REGION Network 51: Step[650] : Transfer PP Left Clamp Open
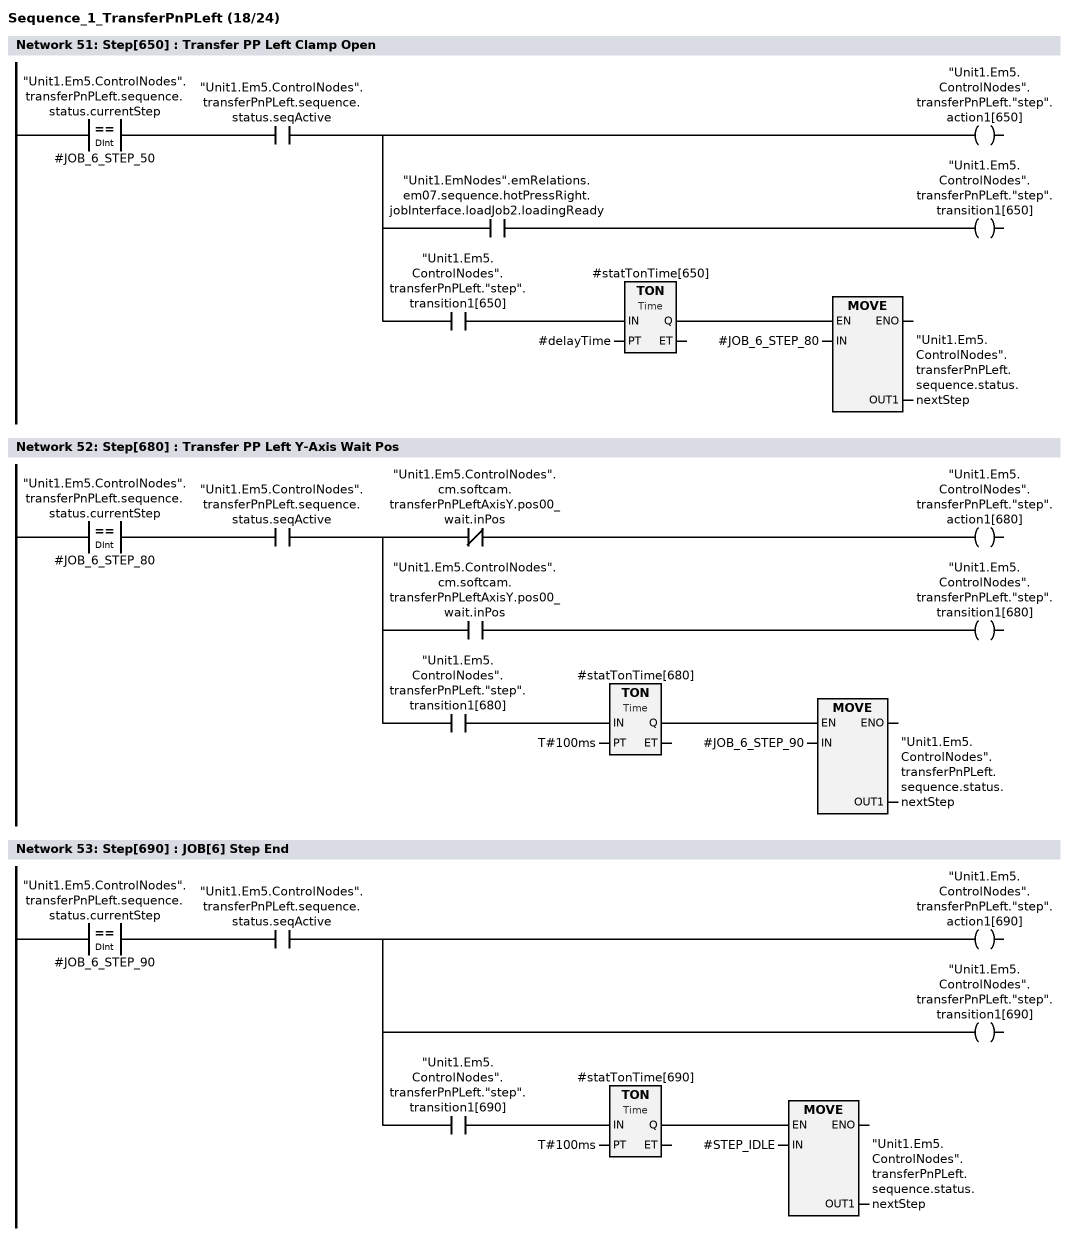
   RUNG wire#powerrail
      { S7_Templates := "SrcType := DInt" } EQ_Contact(in1 := "Unit1.Em5.ControlNodes".transferPnPLeft.sequence.status.currentStep, in2 := #JOB_6_STEP_50)
      Contact( "Unit1.Em5.ControlNodes".transferPnPLeft.sequence.status.seqActive )
      wire#w1
      Coil( "Unit1.Em5.ControlNodes".transferPnPLeft."step".action1[650] )
   END_RUNG
   RUNG wire#w1
      Contact( "Unit1.EmNodes".emRelations.em07.sequence.hotPressRight.jobInterface.loadJob2.loadingReady )
      Coil( "Unit1.Em5.ControlNodes".transferPnPLeft."step".transition1[650] )
   END_RUNG
   RUNG wire#w1
      Contact( "Unit1.Em5.ControlNodes".transferPnPLeft."step".transition1[650] )
      { S7_Templates := "time_type := Time" } #statTonTime[650].TON(pt := #delayTime, et =>)
      Move(in := #JOB_6_STEP_80, out1 => "Unit1.Em5.ControlNodes".transferPnPLeft.sequence.status.nextStep)
   END_RUNG
   // the same network as SCL:
   "Unit1.Em5.ControlNodes".transferPnPLeft."step".action1[650] := ("Unit1.Em5.ControlNodes".transferPnPLeft.sequence.status.currentStep = #JOB_6_STEP_50) AND "Unit1.Em5.ControlNodes".transferPnPLeft.sequence.status.seqActive;
   "Unit1.Em5.ControlNodes".transferPnPLeft."step".transition1[650] := ("Unit1.Em5.ControlNodes".transferPnPLeft.sequence.status.currentStep = #JOB_6_STEP_50) AND "Unit1.Em5.ControlNodes".transferPnPLeft.sequence.status.seqActive AND "Unit1.EmNodes".emRelations.em07.sequence.hotPressRight.jobInterface.loadJob2.loadingReady;
   #statTonTime[650].TON(IN := ("Unit1.Em5.ControlNodes".transferPnPLeft.sequence.status.currentStep = #JOB_6_STEP_50) AND "Unit1.Em5.ControlNodes".transferPnPLeft.sequence.status.seqActive AND "Unit1.Em5.ControlNodes".transferPnPLeft."step".transition1[650],
                         PT := #delayTime);
   IF #statTonTime[650].Q THEN
       "Unit1.Em5.ControlNodes".transferPnPLeft.sequence.status.nextStep := #JOB_6_STEP_80;
   END_IF;
END_REGION

REGION Network 52: Step[680] : Transfer PP Left Y-Axis Wait Pos
   RUNG wire#powerrail
      { S7_Templates := "SrcType := DInt" } EQ_Contact(in1 := "Unit1.Em5.ControlNodes".transferPnPLeft.sequence.status.currentStep, in2 := #JOB_6_STEP_80)
      Contact( "Unit1.Em5.ControlNodes".transferPnPLeft.sequence.status.seqActive )
      wire#w1
      I_Contact( "Unit1.Em5.ControlNodes".cm.softcam.transferPnPLeftAxisY.pos00_wait.inPos )
      Coil( "Unit1.Em5.ControlNodes".transferPnPLeft."step".action1[680] )
   END_RUNG
   RUNG wire#w1
      Contact( "Unit1.Em5.ControlNodes".cm.softcam.transferPnPLeftAxisY.pos00_wait.inPos )
      Coil( "Unit1.Em5.ControlNodes".transferPnPLeft."step".transition1[680] )
   END_RUNG
   RUNG wire#w1
      Contact( "Unit1.Em5.ControlNodes".transferPnPLeft."step".transition1[680] )
      { S7_Templates := "time_type := Time" } #statTonTime[680].TON(pt := T#100ms, et =>)
      Move(in := #JOB_6_STEP_90, out1 => "Unit1.Em5.ControlNodes".transferPnPLeft.sequence.status.nextStep)
   END_RUNG
   // the same network as SCL:
   #_w1 := ("Unit1.Em5.ControlNodes".transferPnPLeft.sequence.status.currentStep = #JOB_6_STEP_80) AND "Unit1.Em5.ControlNodes".transferPnPLeft.sequence.status.seqActive;
   "Unit1.Em5.ControlNodes".transferPnPLeft."step".action1[680] := #_w1 AND NOT "Unit1.Em5.ControlNodes".cm.softcam.transferPnPLeftAxisY.pos00_wait.inPos;
   "Unit1.Em5.ControlNodes".transferPnPLeft."step".transition1[680] := #_w1 AND "Unit1.Em5.ControlNodes".cm.softcam.transferPnPLeftAxisY.pos00_wait.inPos;
   #statTonTime[680].TON(IN := #_w1 AND "Unit1.Em5.ControlNodes".transferPnPLeft."step".transition1[680],
                         PT := T#100ms);
   IF #statTonTime[680].Q THEN
       "Unit1.Em5.ControlNodes".transferPnPLeft.sequence.status.nextStep := #JOB_6_STEP_90;
   END_IF;
END_REGION

REGION Network 53: Step[690] : JOB[6] Step End
   RUNG wire#powerrail
      { S7_Templates := "SrcType := DInt" } EQ_Contact(in1 := "Unit1.Em5.ControlNodes".transferPnPLeft.sequence.status.currentStep, in2 := #JOB_6_STEP_90)
      Contact( "Unit1.Em5.ControlNodes".transferPnPLeft.sequence.status.seqActive )
      wire#w1
      Coil( "Unit1.Em5.ControlNodes".transferPnPLeft."step".action1[690] )
   END_RUNG
   RUNG wire#w1
      Coil( "Unit1.Em5.ControlNodes".transferPnPLeft."step".transition1[690] )
   END_RUNG
   RUNG wire#w1
      Contact( "Unit1.Em5.ControlNodes".transferPnPLeft."step".transition1[690] )
      { S7_Templates := "time_type := Time" } #statTonTime[690].TON(pt := T#100ms, et =>)
      Move(in := #STEP_IDLE, out1 => "Unit1.Em5.ControlNodes".transferPnPLeft.sequence.status.nextStep)
   END_RUNG
   // the same network as SCL:
   "Unit1.Em5.ControlNodes".transferPnPLeft."step".action1[690] := ("Unit1.Em5.ControlNodes".transferPnPLeft.sequence.status.currentStep = #JOB_6_STEP_90) AND "Unit1.Em5.ControlNodes".transferPnPLeft.sequence.status.seqActive;
   "Unit1.Em5.ControlNodes".transferPnPLeft."step".transition1[690] := ("Unit1.Em5.ControlNodes".transferPnPLeft.sequence.status.currentStep = #JOB_6_STEP_90) AND "Unit1.Em5.ControlNodes".transferPnPLeft.sequence.status.seqActive;
   #statTonTime[690].TON(IN := ("Unit1.Em5.ControlNodes".transferPnPLeft.sequence.status.currentStep = #JOB_6_STEP_90) AND "Unit1.Em5.ControlNodes".transferPnPLeft.sequence.status.seqActive AND "Unit1.Em5.ControlNodes".transferPnPLeft."step".transition1[690],
                         PT := T#100ms);
   IF #statTonTime[690].Q THEN
       "Unit1.Em5.ControlNodes".transferPnPLeft.sequence.status.nextStep := #STEP_IDLE;
   END_IF;
END_REGION

REGION Network 54: *********** JOB[7] HOT PRESS RIGHT JR GET=AUTO-[B] *************
END_REGION

REGION Network 55: Step[701] : JOB[7] Condition
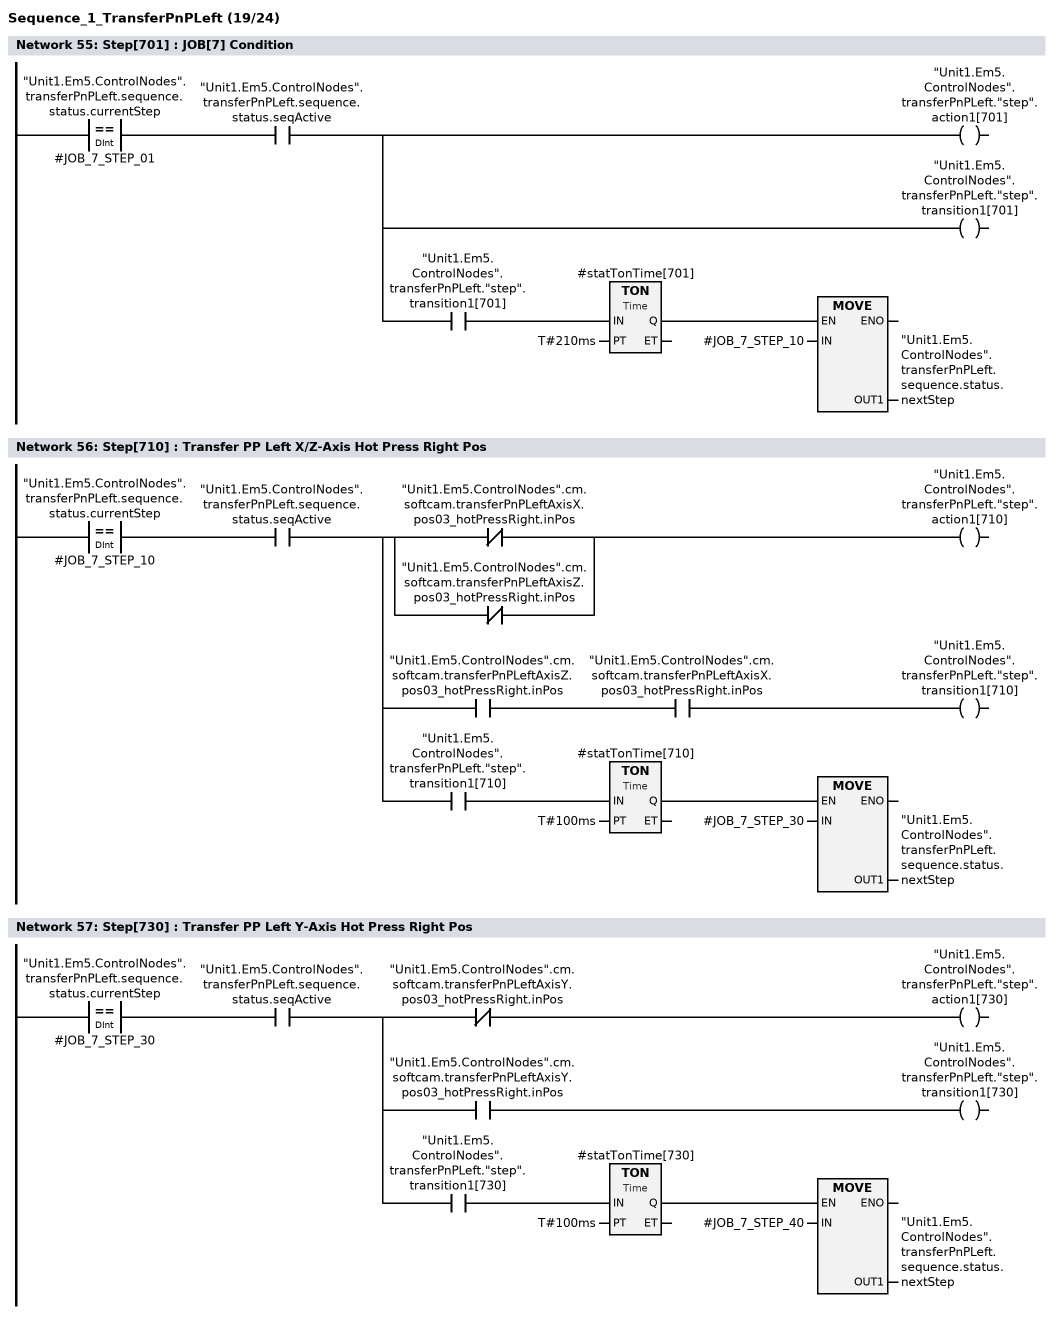
   RUNG wire#powerrail
      { S7_Templates := "SrcType := DInt" } EQ_Contact(in1 := "Unit1.Em5.ControlNodes".transferPnPLeft.sequence.status.currentStep, in2 := #JOB_7_STEP_01)
      Contact( "Unit1.Em5.ControlNodes".transferPnPLeft.sequence.status.seqActive )
      wire#w1
      Coil( "Unit1.Em5.ControlNodes".transferPnPLeft."step".action1[701] )
   END_RUNG
   RUNG wire#w1
      Coil( "Unit1.Em5.ControlNodes".transferPnPLeft."step".transition1[701] )
   END_RUNG
   RUNG wire#w1
      Contact( "Unit1.Em5.ControlNodes".transferPnPLeft."step".transition1[701] )
      { S7_Templates := "time_type := Time" } #statTonTime[701].TON(pt := T#210ms, et =>)
      Move(in := #JOB_7_STEP_10, out1 => "Unit1.Em5.ControlNodes".transferPnPLeft.sequence.status.nextStep)
   END_RUNG
   // the same network as SCL:
   "Unit1.Em5.ControlNodes".transferPnPLeft."step".action1[701] := ("Unit1.Em5.ControlNodes".transferPnPLeft.sequence.status.currentStep = #JOB_7_STEP_01) AND "Unit1.Em5.ControlNodes".transferPnPLeft.sequence.status.seqActive;
   "Unit1.Em5.ControlNodes".transferPnPLeft."step".transition1[701] := ("Unit1.Em5.ControlNodes".transferPnPLeft.sequence.status.currentStep = #JOB_7_STEP_01) AND "Unit1.Em5.ControlNodes".transferPnPLeft.sequence.status.seqActive;
   #statTonTime[701].TON(IN := ("Unit1.Em5.ControlNodes".transferPnPLeft.sequence.status.currentStep = #JOB_7_STEP_01) AND "Unit1.Em5.ControlNodes".transferPnPLeft.sequence.status.seqActive AND "Unit1.Em5.ControlNodes".transferPnPLeft."step".transition1[701],
                         PT := T#210ms);
   IF #statTonTime[701].Q THEN
       "Unit1.Em5.ControlNodes".transferPnPLeft.sequence.status.nextStep := #JOB_7_STEP_10;
   END_IF;
END_REGION

REGION Network 56: Step[710] : Transfer PP Left X/Z-Axis Hot Press Right Pos
   RUNG wire#powerrail
      { S7_Templates := "SrcType := DInt" } EQ_Contact(in1 := "Unit1.Em5.ControlNodes".transferPnPLeft.sequence.status.currentStep, in2 := #JOB_7_STEP_10)
      Contact( "Unit1.Em5.ControlNodes".transferPnPLeft.sequence.status.seqActive )
      wire#w1
      I_Contact( "Unit1.Em5.ControlNodes".cm.softcam.transferPnPLeftAxisX.pos03_hotPressRight.inPos )
      wire#w2
      Coil( "Unit1.Em5.ControlNodes".transferPnPLeft."step".action1[710] )
   END_RUNG
   RUNG wire#w1
      I_Contact( "Unit1.Em5.ControlNodes".cm.softcam.transferPnPLeftAxisZ.pos03_hotPressRight.inPos )
   END_RUNG wire#w2
   RUNG wire#w1
      Contact( "Unit1.Em5.ControlNodes".cm.softcam.transferPnPLeftAxisZ.pos03_hotPressRight.inPos )
      Contact( "Unit1.Em5.ControlNodes".cm.softcam.transferPnPLeftAxisX.pos03_hotPressRight.inPos )
      Coil( "Unit1.Em5.ControlNodes".transferPnPLeft."step".transition1[710] )
   END_RUNG
   RUNG wire#w1
      Contact( "Unit1.Em5.ControlNodes".transferPnPLeft."step".transition1[710] )
      { S7_Templates := "time_type := Time" } #statTonTime[710].TON(pt := T#100ms, et =>)
      Move(in := #JOB_7_STEP_30, out1 => "Unit1.Em5.ControlNodes".transferPnPLeft.sequence.status.nextStep)
   END_RUNG
   // the same network as SCL:
   #_w1 := ("Unit1.Em5.ControlNodes".transferPnPLeft.sequence.status.currentStep = #JOB_7_STEP_10) AND "Unit1.Em5.ControlNodes".transferPnPLeft.sequence.status.seqActive;
   "Unit1.Em5.ControlNodes".transferPnPLeft."step".action1[710] := #_w1 AND (NOT "Unit1.Em5.ControlNodes".cm.softcam.transferPnPLeftAxisX.pos03_hotPressRight.inPos OR NOT "Unit1.Em5.ControlNodes".cm.softcam.transferPnPLeftAxisZ.pos03_hotPressRight.inPos);
   "Unit1.Em5.ControlNodes".transferPnPLeft."step".transition1[710] := #_w1 AND "Unit1.Em5.ControlNodes".cm.softcam.transferPnPLeftAxisZ.pos03_hotPressRight.inPos AND "Unit1.Em5.ControlNodes".cm.softcam.transferPnPLeftAxisX.pos03_hotPressRight.inPos;
   #statTonTime[710].TON(IN := #_w1 AND "Unit1.Em5.ControlNodes".transferPnPLeft."step".transition1[710],
                         PT := T#100ms);
   IF #statTonTime[710].Q THEN
       "Unit1.Em5.ControlNodes".transferPnPLeft.sequence.status.nextStep := #JOB_7_STEP_30;
   END_IF;
END_REGION

REGION Network 57: Step[730] : Transfer PP Left Y-Axis Hot Press Right Pos
   RUNG wire#powerrail
      { S7_Templates := "SrcType := DInt" } EQ_Contact(in1 := "Unit1.Em5.ControlNodes".transferPnPLeft.sequence.status.currentStep, in2 := #JOB_7_STEP_30)
      Contact( "Unit1.Em5.ControlNodes".transferPnPLeft.sequence.status.seqActive )
      wire#w1
      I_Contact( "Unit1.Em5.ControlNodes".cm.softcam.transferPnPLeftAxisY.pos03_hotPressRight.inPos )
      Coil( "Unit1.Em5.ControlNodes".transferPnPLeft."step".action1[730] )
   END_RUNG
   RUNG wire#w1
      Contact( "Unit1.Em5.ControlNodes".cm.softcam.transferPnPLeftAxisY.pos03_hotPressRight.inPos )
      Coil( "Unit1.Em5.ControlNodes".transferPnPLeft."step".transition1[730] )
   END_RUNG
   RUNG wire#w1
      Contact( "Unit1.Em5.ControlNodes".transferPnPLeft."step".transition1[730] )
      { S7_Templates := "time_type := Time" } #statTonTime[730].TON(pt := T#100ms, et =>)
      Move(in := #JOB_7_STEP_40, out1 => "Unit1.Em5.ControlNodes".transferPnPLeft.sequence.status.nextStep)
   END_RUNG
   // the same network as SCL:
   #_w1 := ("Unit1.Em5.ControlNodes".transferPnPLeft.sequence.status.currentStep = #JOB_7_STEP_30) AND "Unit1.Em5.ControlNodes".transferPnPLeft.sequence.status.seqActive;
   "Unit1.Em5.ControlNodes".transferPnPLeft."step".action1[730] := #_w1 AND NOT "Unit1.Em5.ControlNodes".cm.softcam.transferPnPLeftAxisY.pos03_hotPressRight.inPos;
   "Unit1.Em5.ControlNodes".transferPnPLeft."step".transition1[730] := #_w1 AND "Unit1.Em5.ControlNodes".cm.softcam.transferPnPLeftAxisY.pos03_hotPressRight.inPos;
   #statTonTime[730].TON(IN := #_w1 AND "Unit1.Em5.ControlNodes".transferPnPLeft."step".transition1[730],
                         PT := T#100ms);
   IF #statTonTime[730].Q THEN
       "Unit1.Em5.ControlNodes".transferPnPLeft.sequence.status.nextStep := #JOB_7_STEP_40;
   END_IF;
END_REGION

REGION Network 58: Step[740] : Transfer PP Left Clamp Close
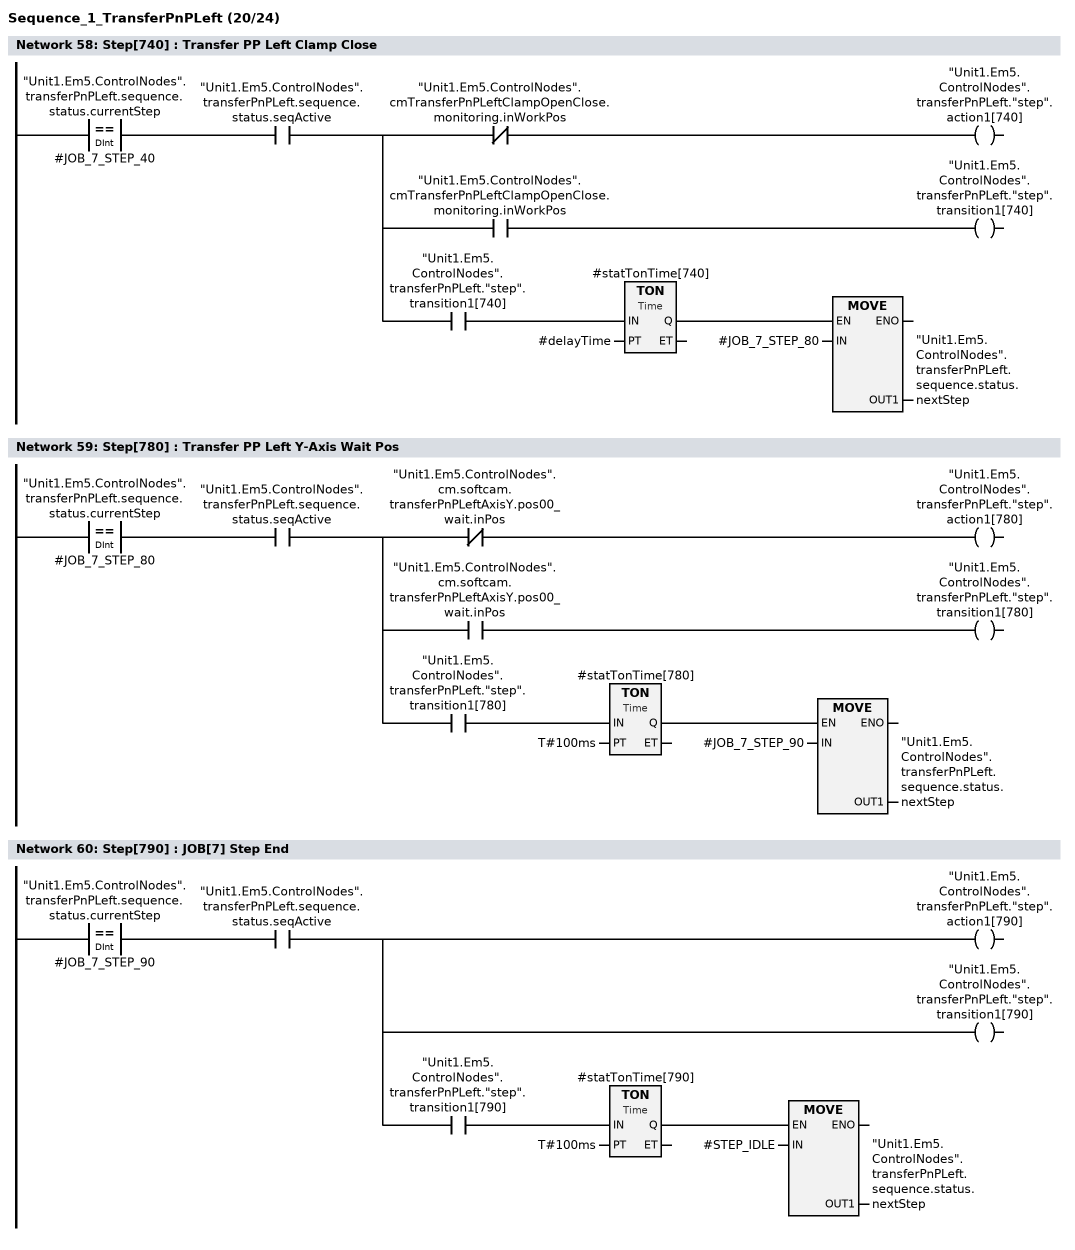
   RUNG wire#powerrail
      { S7_Templates := "SrcType := DInt" } EQ_Contact(in1 := "Unit1.Em5.ControlNodes".transferPnPLeft.sequence.status.currentStep, in2 := #JOB_7_STEP_40)
      Contact( "Unit1.Em5.ControlNodes".transferPnPLeft.sequence.status.seqActive )
      wire#w1
      I_Contact( "Unit1.Em5.ControlNodes".cmTransferPnPLeftClampOpenClose.monitoring.inWorkPos )
      Coil( "Unit1.Em5.ControlNodes".transferPnPLeft."step".action1[740] )
   END_RUNG
   RUNG wire#w1
      Contact( "Unit1.Em5.ControlNodes".cmTransferPnPLeftClampOpenClose.monitoring.inWorkPos )
      Coil( "Unit1.Em5.ControlNodes".transferPnPLeft."step".transition1[740] )
   END_RUNG
   RUNG wire#w1
      Contact( "Unit1.Em5.ControlNodes".transferPnPLeft."step".transition1[740] )
      { S7_Templates := "time_type := Time" } #statTonTime[740].TON(pt := #delayTime, et =>)
      Move(in := #JOB_7_STEP_80, out1 => "Unit1.Em5.ControlNodes".transferPnPLeft.sequence.status.nextStep)
   END_RUNG
   // the same network as SCL:
   #_w1 := ("Unit1.Em5.ControlNodes".transferPnPLeft.sequence.status.currentStep = #JOB_7_STEP_40) AND "Unit1.Em5.ControlNodes".transferPnPLeft.sequence.status.seqActive;
   "Unit1.Em5.ControlNodes".transferPnPLeft."step".action1[740] := #_w1 AND NOT "Unit1.Em5.ControlNodes".cmTransferPnPLeftClampOpenClose.monitoring.inWorkPos;
   "Unit1.Em5.ControlNodes".transferPnPLeft."step".transition1[740] := #_w1 AND "Unit1.Em5.ControlNodes".cmTransferPnPLeftClampOpenClose.monitoring.inWorkPos;
   #statTonTime[740].TON(IN := #_w1 AND "Unit1.Em5.ControlNodes".transferPnPLeft."step".transition1[740],
                         PT := #delayTime);
   IF #statTonTime[740].Q THEN
       "Unit1.Em5.ControlNodes".transferPnPLeft.sequence.status.nextStep := #JOB_7_STEP_80;
   END_IF;
END_REGION

REGION Network 59: Step[780] : Transfer PP Left Y-Axis Wait Pos
   RUNG wire#powerrail
      { S7_Templates := "SrcType := DInt" } EQ_Contact(in1 := "Unit1.Em5.ControlNodes".transferPnPLeft.sequence.status.currentStep, in2 := #JOB_7_STEP_80)
      Contact( "Unit1.Em5.ControlNodes".transferPnPLeft.sequence.status.seqActive )
      wire#w1
      I_Contact( "Unit1.Em5.ControlNodes".cm.softcam.transferPnPLeftAxisY.pos00_wait.inPos )
      Coil( "Unit1.Em5.ControlNodes".transferPnPLeft."step".action1[780] )
   END_RUNG
   RUNG wire#w1
      Contact( "Unit1.Em5.ControlNodes".cm.softcam.transferPnPLeftAxisY.pos00_wait.inPos )
      Coil( "Unit1.Em5.ControlNodes".transferPnPLeft."step".transition1[780] )
   END_RUNG
   RUNG wire#w1
      Contact( "Unit1.Em5.ControlNodes".transferPnPLeft."step".transition1[780] )
      { S7_Templates := "time_type := Time" } #statTonTime[780].TON(pt := T#100ms, et =>)
      Move(in := #JOB_7_STEP_90, out1 => "Unit1.Em5.ControlNodes".transferPnPLeft.sequence.status.nextStep)
   END_RUNG
   // the same network as SCL:
   #_w1 := ("Unit1.Em5.ControlNodes".transferPnPLeft.sequence.status.currentStep = #JOB_7_STEP_80) AND "Unit1.Em5.ControlNodes".transferPnPLeft.sequence.status.seqActive;
   "Unit1.Em5.ControlNodes".transferPnPLeft."step".action1[780] := #_w1 AND NOT "Unit1.Em5.ControlNodes".cm.softcam.transferPnPLeftAxisY.pos00_wait.inPos;
   "Unit1.Em5.ControlNodes".transferPnPLeft."step".transition1[780] := #_w1 AND "Unit1.Em5.ControlNodes".cm.softcam.transferPnPLeftAxisY.pos00_wait.inPos;
   #statTonTime[780].TON(IN := #_w1 AND "Unit1.Em5.ControlNodes".transferPnPLeft."step".transition1[780],
                         PT := T#100ms);
   IF #statTonTime[780].Q THEN
       "Unit1.Em5.ControlNodes".transferPnPLeft.sequence.status.nextStep := #JOB_7_STEP_90;
   END_IF;
END_REGION

REGION Network 60: Step[790] : JOB[7] Step End
   RUNG wire#powerrail
      { S7_Templates := "SrcType := DInt" } EQ_Contact(in1 := "Unit1.Em5.ControlNodes".transferPnPLeft.sequence.status.currentStep, in2 := #JOB_7_STEP_90)
      Contact( "Unit1.Em5.ControlNodes".transferPnPLeft.sequence.status.seqActive )
      wire#w1
      Coil( "Unit1.Em5.ControlNodes".transferPnPLeft."step".action1[790] )
   END_RUNG
   RUNG wire#w1
      Coil( "Unit1.Em5.ControlNodes".transferPnPLeft."step".transition1[790] )
   END_RUNG
   RUNG wire#w1
      Contact( "Unit1.Em5.ControlNodes".transferPnPLeft."step".transition1[790] )
      { S7_Templates := "time_type := Time" } #statTonTime[790].TON(pt := T#100ms, et =>)
      Move(in := #STEP_IDLE, out1 => "Unit1.Em5.ControlNodes".transferPnPLeft.sequence.status.nextStep)
   END_RUNG
   // the same network as SCL:
   "Unit1.Em5.ControlNodes".transferPnPLeft."step".action1[790] := ("Unit1.Em5.ControlNodes".transferPnPLeft.sequence.status.currentStep = #JOB_7_STEP_90) AND "Unit1.Em5.ControlNodes".transferPnPLeft.sequence.status.seqActive;
   "Unit1.Em5.ControlNodes".transferPnPLeft."step".transition1[790] := ("Unit1.Em5.ControlNodes".transferPnPLeft.sequence.status.currentStep = #JOB_7_STEP_90) AND "Unit1.Em5.ControlNodes".transferPnPLeft.sequence.status.seqActive;
   #statTonTime[790].TON(IN := ("Unit1.Em5.ControlNodes".transferPnPLeft.sequence.status.currentStep = #JOB_7_STEP_90) AND "Unit1.Em5.ControlNodes".transferPnPLeft.sequence.status.seqActive AND "Unit1.Em5.ControlNodes".transferPnPLeft."step".transition1[790],
                         PT := T#100ms);
   IF #statTonTime[790].Q THEN
       "Unit1.Em5.ControlNodes".transferPnPLeft.sequence.status.nextStep := #STEP_IDLE;
   END_IF;
END_REGION

REGION Network 61: *********** JOB[9] HIPOT & THICKNESS JR PUT=AUTO-[A][B] ************
END_REGION

REGION Network 62: Step[901] : JOB[9] Condition
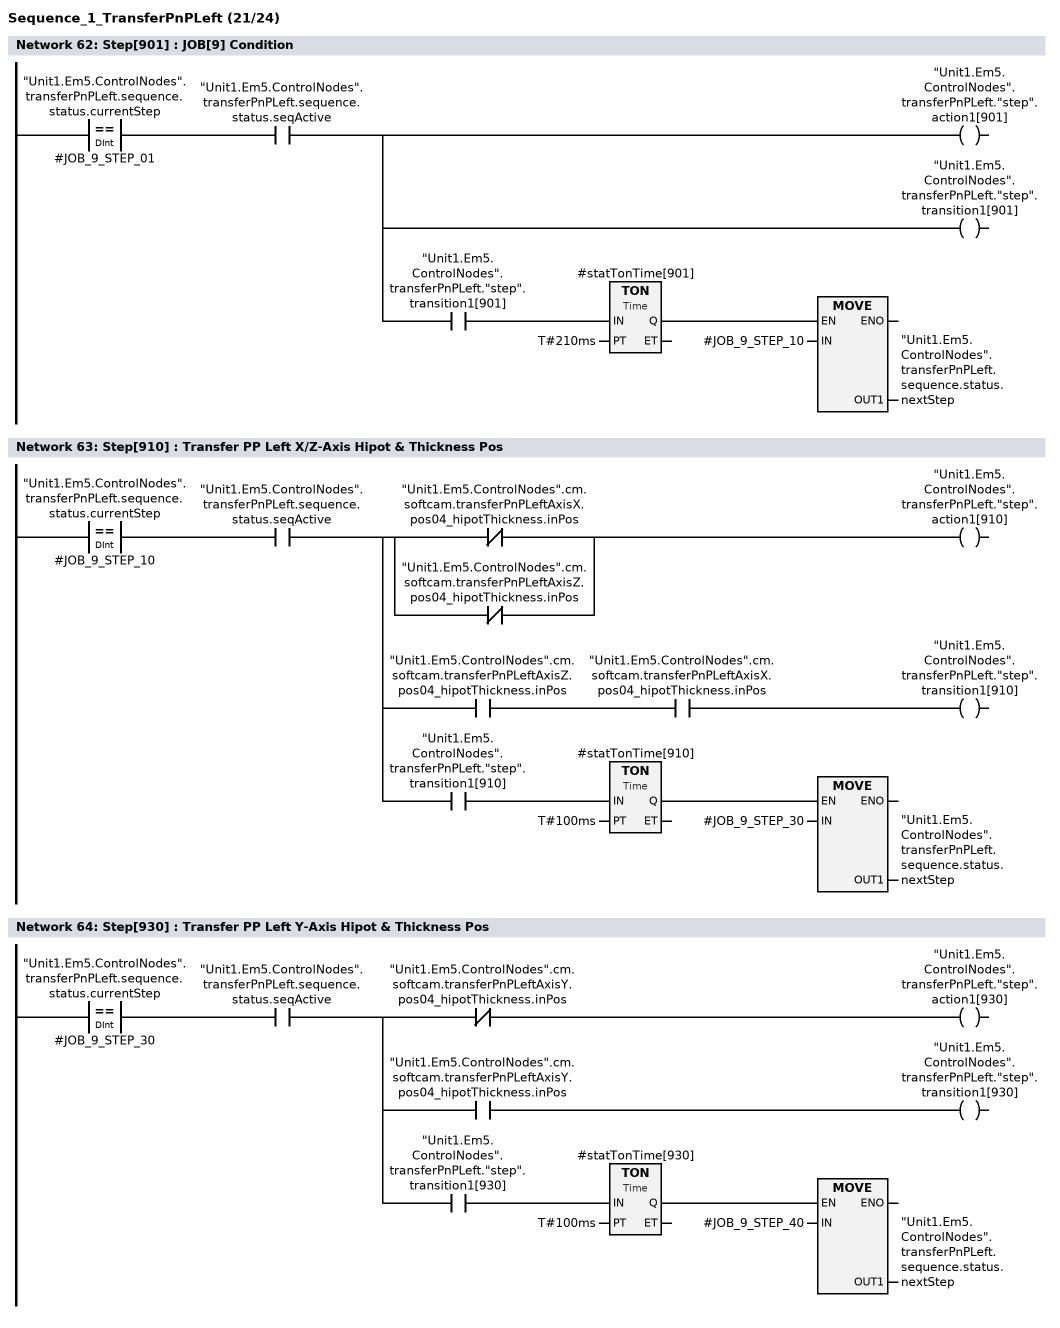
   RUNG wire#powerrail
      { S7_Templates := "SrcType := DInt" } EQ_Contact(in1 := "Unit1.Em5.ControlNodes".transferPnPLeft.sequence.status.currentStep, in2 := #JOB_9_STEP_01)
      Contact( "Unit1.Em5.ControlNodes".transferPnPLeft.sequence.status.seqActive )
      wire#w1
      Coil( "Unit1.Em5.ControlNodes".transferPnPLeft."step".action1[901] )
   END_RUNG
   RUNG wire#w1
      Coil( "Unit1.Em5.ControlNodes".transferPnPLeft."step".transition1[901] )
   END_RUNG
   RUNG wire#w1
      Contact( "Unit1.Em5.ControlNodes".transferPnPLeft."step".transition1[901] )
      { S7_Templates := "time_type := Time" } #statTonTime[901].TON(pt := T#210ms, et =>)
      Move(in := #JOB_9_STEP_10, out1 => "Unit1.Em5.ControlNodes".transferPnPLeft.sequence.status.nextStep)
   END_RUNG
   // the same network as SCL:
   "Unit1.Em5.ControlNodes".transferPnPLeft."step".action1[901] := ("Unit1.Em5.ControlNodes".transferPnPLeft.sequence.status.currentStep = #JOB_9_STEP_01) AND "Unit1.Em5.ControlNodes".transferPnPLeft.sequence.status.seqActive;
   "Unit1.Em5.ControlNodes".transferPnPLeft."step".transition1[901] := ("Unit1.Em5.ControlNodes".transferPnPLeft.sequence.status.currentStep = #JOB_9_STEP_01) AND "Unit1.Em5.ControlNodes".transferPnPLeft.sequence.status.seqActive;
   #statTonTime[901].TON(IN := ("Unit1.Em5.ControlNodes".transferPnPLeft.sequence.status.currentStep = #JOB_9_STEP_01) AND "Unit1.Em5.ControlNodes".transferPnPLeft.sequence.status.seqActive AND "Unit1.Em5.ControlNodes".transferPnPLeft."step".transition1[901],
                         PT := T#210ms);
   IF #statTonTime[901].Q THEN
       "Unit1.Em5.ControlNodes".transferPnPLeft.sequence.status.nextStep := #JOB_9_STEP_10;
   END_IF;
END_REGION

REGION Network 63: Step[910] : Transfer PP Left X/Z-Axis Hipot & Thickness Pos
   RUNG wire#powerrail
      { S7_Templates := "SrcType := DInt" } EQ_Contact(in1 := "Unit1.Em5.ControlNodes".transferPnPLeft.sequence.status.currentStep, in2 := #JOB_9_STEP_10)
      Contact( "Unit1.Em5.ControlNodes".transferPnPLeft.sequence.status.seqActive )
      wire#w1
      I_Contact( "Unit1.Em5.ControlNodes".cm.softcam.transferPnPLeftAxisX.pos04_hipotThickness.inPos )
      wire#w2
      Coil( "Unit1.Em5.ControlNodes".transferPnPLeft."step".action1[910] )
   END_RUNG
   RUNG wire#w1
      I_Contact( "Unit1.Em5.ControlNodes".cm.softcam.transferPnPLeftAxisZ.pos04_hipotThickness.inPos )
   END_RUNG wire#w2
   RUNG wire#w1
      Contact( "Unit1.Em5.ControlNodes".cm.softcam.transferPnPLeftAxisZ.pos04_hipotThickness.inPos )
      Contact( "Unit1.Em5.ControlNodes".cm.softcam.transferPnPLeftAxisX.pos04_hipotThickness.inPos )
      Coil( "Unit1.Em5.ControlNodes".transferPnPLeft."step".transition1[910] )
   END_RUNG
   RUNG wire#w1
      Contact( "Unit1.Em5.ControlNodes".transferPnPLeft."step".transition1[910] )
      { S7_Templates := "time_type := Time" } #statTonTime[910].TON(pt := T#100ms, et =>)
      Move(in := #JOB_9_STEP_30, out1 => "Unit1.Em5.ControlNodes".transferPnPLeft.sequence.status.nextStep)
   END_RUNG
   // the same network as SCL:
   #_w1 := ("Unit1.Em5.ControlNodes".transferPnPLeft.sequence.status.currentStep = #JOB_9_STEP_10) AND "Unit1.Em5.ControlNodes".transferPnPLeft.sequence.status.seqActive;
   "Unit1.Em5.ControlNodes".transferPnPLeft."step".action1[910] := #_w1 AND (NOT "Unit1.Em5.ControlNodes".cm.softcam.transferPnPLeftAxisX.pos04_hipotThickness.inPos OR NOT "Unit1.Em5.ControlNodes".cm.softcam.transferPnPLeftAxisZ.pos04_hipotThickness.inPos);
   "Unit1.Em5.ControlNodes".transferPnPLeft."step".transition1[910] := #_w1 AND "Unit1.Em5.ControlNodes".cm.softcam.transferPnPLeftAxisZ.pos04_hipotThickness.inPos AND "Unit1.Em5.ControlNodes".cm.softcam.transferPnPLeftAxisX.pos04_hipotThickness.inPos;
   #statTonTime[910].TON(IN := #_w1 AND "Unit1.Em5.ControlNodes".transferPnPLeft."step".transition1[910],
                         PT := T#100ms);
   IF #statTonTime[910].Q THEN
       "Unit1.Em5.ControlNodes".transferPnPLeft.sequence.status.nextStep := #JOB_9_STEP_30;
   END_IF;
END_REGION

REGION Network 64: Step[930] : Transfer PP Left Y-Axis Hipot & Thickness Pos
   RUNG wire#powerrail
      { S7_Templates := "SrcType := DInt" } EQ_Contact(in1 := "Unit1.Em5.ControlNodes".transferPnPLeft.sequence.status.currentStep, in2 := #JOB_9_STEP_30)
      Contact( "Unit1.Em5.ControlNodes".transferPnPLeft.sequence.status.seqActive )
      wire#w1
      I_Contact( "Unit1.Em5.ControlNodes".cm.softcam.transferPnPLeftAxisY.pos04_hipotThickness.inPos )
      Coil( "Unit1.Em5.ControlNodes".transferPnPLeft."step".action1[930] )
   END_RUNG
   RUNG wire#w1
      Contact( "Unit1.Em5.ControlNodes".cm.softcam.transferPnPLeftAxisY.pos04_hipotThickness.inPos )
      Coil( "Unit1.Em5.ControlNodes".transferPnPLeft."step".transition1[930] )
   END_RUNG
   RUNG wire#w1
      Contact( "Unit1.Em5.ControlNodes".transferPnPLeft."step".transition1[930] )
      { S7_Templates := "time_type := Time" } #statTonTime[930].TON(pt := T#100ms, et =>)
      Move(in := #JOB_9_STEP_40, out1 => "Unit1.Em5.ControlNodes".transferPnPLeft.sequence.status.nextStep)
   END_RUNG
   // the same network as SCL:
   #_w1 := ("Unit1.Em5.ControlNodes".transferPnPLeft.sequence.status.currentStep = #JOB_9_STEP_30) AND "Unit1.Em5.ControlNodes".transferPnPLeft.sequence.status.seqActive;
   "Unit1.Em5.ControlNodes".transferPnPLeft."step".action1[930] := #_w1 AND NOT "Unit1.Em5.ControlNodes".cm.softcam.transferPnPLeftAxisY.pos04_hipotThickness.inPos;
   "Unit1.Em5.ControlNodes".transferPnPLeft."step".transition1[930] := #_w1 AND "Unit1.Em5.ControlNodes".cm.softcam.transferPnPLeftAxisY.pos04_hipotThickness.inPos;
   #statTonTime[930].TON(IN := #_w1 AND "Unit1.Em5.ControlNodes".transferPnPLeft."step".transition1[930],
                         PT := T#100ms);
   IF #statTonTime[930].Q THEN
       "Unit1.Em5.ControlNodes".transferPnPLeft.sequence.status.nextStep := #JOB_9_STEP_40;
   END_IF;
END_REGION

REGION Network 65: Step[940] : Transfer PP Left [Lift Up Request] => Hipot & Thickness
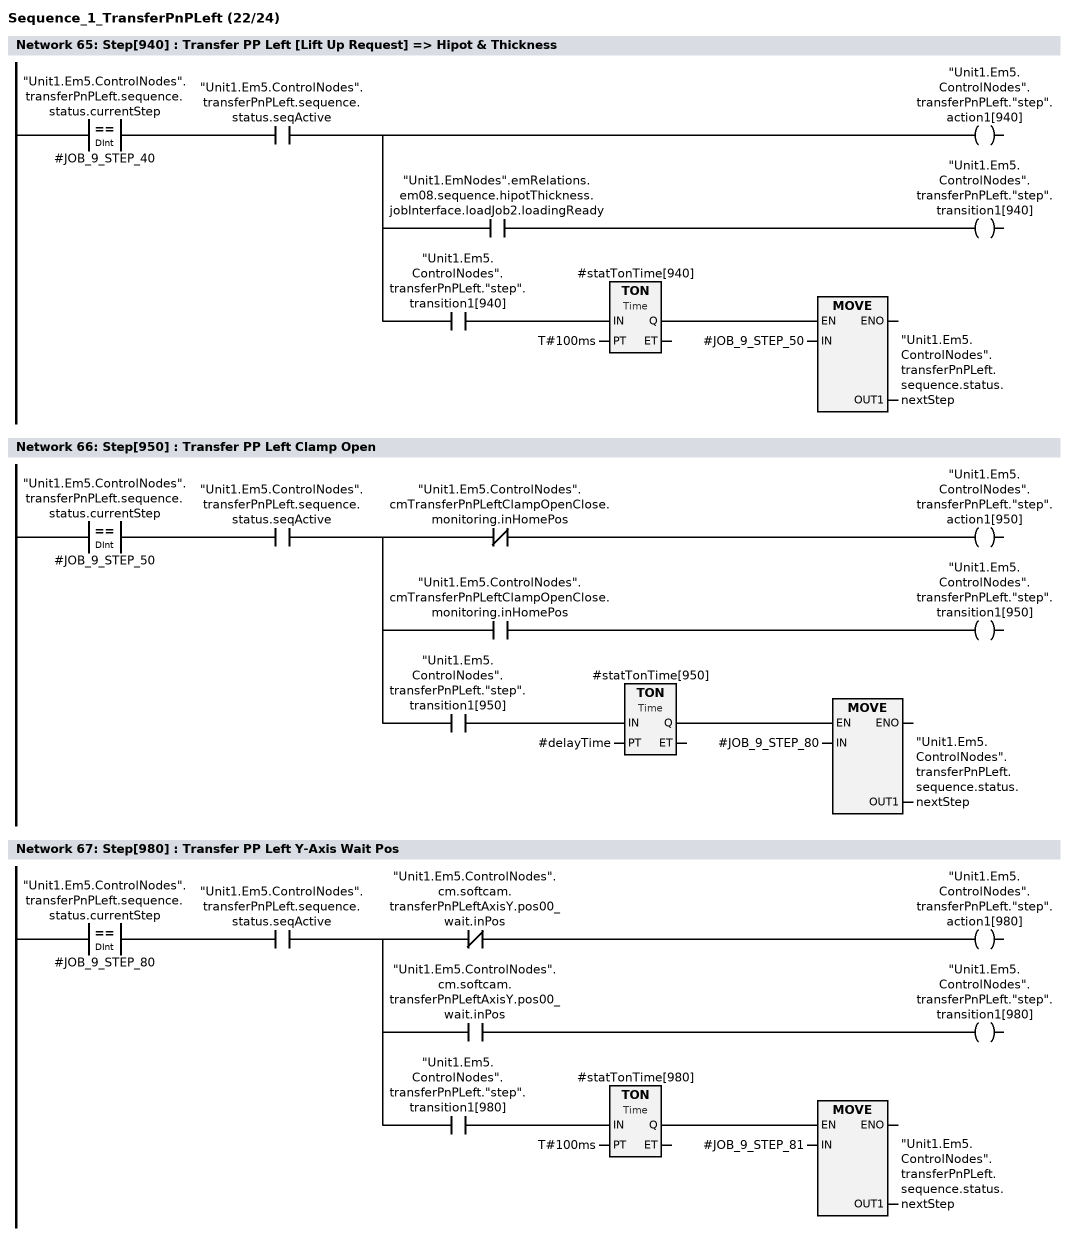
   RUNG wire#powerrail
      { S7_Templates := "SrcType := DInt" } EQ_Contact(in1 := "Unit1.Em5.ControlNodes".transferPnPLeft.sequence.status.currentStep, in2 := #JOB_9_STEP_40)
      Contact( "Unit1.Em5.ControlNodes".transferPnPLeft.sequence.status.seqActive )
      wire#w1
      Coil( "Unit1.Em5.ControlNodes".transferPnPLeft."step".action1[940] )
   END_RUNG
   RUNG wire#w1
      Contact( "Unit1.EmNodes".emRelations.em08.sequence.hipotThickness.jobInterface.loadJob2.loadingReady )
      Coil( "Unit1.Em5.ControlNodes".transferPnPLeft."step".transition1[940] )
   END_RUNG
   RUNG wire#w1
      Contact( "Unit1.Em5.ControlNodes".transferPnPLeft."step".transition1[940] )
      { S7_Templates := "time_type := Time" } #statTonTime[940].TON(pt := T#100ms, et =>)
      Move(in := #JOB_9_STEP_50, out1 => "Unit1.Em5.ControlNodes".transferPnPLeft.sequence.status.nextStep)
   END_RUNG
   // the same network as SCL:
   "Unit1.Em5.ControlNodes".transferPnPLeft."step".action1[940] := ("Unit1.Em5.ControlNodes".transferPnPLeft.sequence.status.currentStep = #JOB_9_STEP_40) AND "Unit1.Em5.ControlNodes".transferPnPLeft.sequence.status.seqActive;
   "Unit1.Em5.ControlNodes".transferPnPLeft."step".transition1[940] := ("Unit1.Em5.ControlNodes".transferPnPLeft.sequence.status.currentStep = #JOB_9_STEP_40) AND "Unit1.Em5.ControlNodes".transferPnPLeft.sequence.status.seqActive AND "Unit1.EmNodes".emRelations.em08.sequence.hipotThickness.jobInterface.loadJob2.loadingReady;
   #statTonTime[940].TON(IN := ("Unit1.Em5.ControlNodes".transferPnPLeft.sequence.status.currentStep = #JOB_9_STEP_40) AND "Unit1.Em5.ControlNodes".transferPnPLeft.sequence.status.seqActive AND "Unit1.Em5.ControlNodes".transferPnPLeft."step".transition1[940],
                         PT := T#100ms);
   IF #statTonTime[940].Q THEN
       "Unit1.Em5.ControlNodes".transferPnPLeft.sequence.status.nextStep := #JOB_9_STEP_50;
   END_IF;
END_REGION

REGION Network 66: Step[950] : Transfer PP Left Clamp Open
   RUNG wire#powerrail
      { S7_Templates := "SrcType := DInt" } EQ_Contact(in1 := "Unit1.Em5.ControlNodes".transferPnPLeft.sequence.status.currentStep, in2 := #JOB_9_STEP_50)
      Contact( "Unit1.Em5.ControlNodes".transferPnPLeft.sequence.status.seqActive )
      wire#w1
      I_Contact( "Unit1.Em5.ControlNodes".cmTransferPnPLeftClampOpenClose.monitoring.inHomePos )
      Coil( "Unit1.Em5.ControlNodes".transferPnPLeft."step".action1[950] )
   END_RUNG
   RUNG wire#w1
      Contact( "Unit1.Em5.ControlNodes".cmTransferPnPLeftClampOpenClose.monitoring.inHomePos )
      Coil( "Unit1.Em5.ControlNodes".transferPnPLeft."step".transition1[950] )
   END_RUNG
   RUNG wire#w1
      Contact( "Unit1.Em5.ControlNodes".transferPnPLeft."step".transition1[950] )
      { S7_Templates := "time_type := Time" } #statTonTime[950].TON(pt := #delayTime, et =>)
      Move(in := #JOB_9_STEP_80, out1 => "Unit1.Em5.ControlNodes".transferPnPLeft.sequence.status.nextStep)
   END_RUNG
   // the same network as SCL:
   #_w1 := ("Unit1.Em5.ControlNodes".transferPnPLeft.sequence.status.currentStep = #JOB_9_STEP_50) AND "Unit1.Em5.ControlNodes".transferPnPLeft.sequence.status.seqActive;
   "Unit1.Em5.ControlNodes".transferPnPLeft."step".action1[950] := #_w1 AND NOT "Unit1.Em5.ControlNodes".cmTransferPnPLeftClampOpenClose.monitoring.inHomePos;
   "Unit1.Em5.ControlNodes".transferPnPLeft."step".transition1[950] := #_w1 AND "Unit1.Em5.ControlNodes".cmTransferPnPLeftClampOpenClose.monitoring.inHomePos;
   #statTonTime[950].TON(IN := #_w1 AND "Unit1.Em5.ControlNodes".transferPnPLeft."step".transition1[950],
                         PT := #delayTime);
   IF #statTonTime[950].Q THEN
       "Unit1.Em5.ControlNodes".transferPnPLeft.sequence.status.nextStep := #JOB_9_STEP_80;
   END_IF;
END_REGION

REGION Network 67: Step[980] : Transfer PP Left Y-Axis Wait Pos
   RUNG wire#powerrail
      { S7_Templates := "SrcType := DInt" } EQ_Contact(in1 := "Unit1.Em5.ControlNodes".transferPnPLeft.sequence.status.currentStep, in2 := #JOB_9_STEP_80)
      Contact( "Unit1.Em5.ControlNodes".transferPnPLeft.sequence.status.seqActive )
      wire#w1
      I_Contact( "Unit1.Em5.ControlNodes".cm.softcam.transferPnPLeftAxisY.pos00_wait.inPos )
      Coil( "Unit1.Em5.ControlNodes".transferPnPLeft."step".action1[980] )
   END_RUNG
   RUNG wire#w1
      Contact( "Unit1.Em5.ControlNodes".cm.softcam.transferPnPLeftAxisY.pos00_wait.inPos )
      Coil( "Unit1.Em5.ControlNodes".transferPnPLeft."step".transition1[980] )
   END_RUNG
   RUNG wire#w1
      Contact( "Unit1.Em5.ControlNodes".transferPnPLeft."step".transition1[980] )
      { S7_Templates := "time_type := Time" } #statTonTime[980].TON(pt := T#100ms, et =>)
      Move(in := #JOB_9_STEP_81, out1 => "Unit1.Em5.ControlNodes".transferPnPLeft.sequence.status.nextStep)
   END_RUNG
   // the same network as SCL:
   #_w1 := ("Unit1.Em5.ControlNodes".transferPnPLeft.sequence.status.currentStep = #JOB_9_STEP_80) AND "Unit1.Em5.ControlNodes".transferPnPLeft.sequence.status.seqActive;
   "Unit1.Em5.ControlNodes".transferPnPLeft."step".action1[980] := #_w1 AND NOT "Unit1.Em5.ControlNodes".cm.softcam.transferPnPLeftAxisY.pos00_wait.inPos;
   "Unit1.Em5.ControlNodes".transferPnPLeft."step".transition1[980] := #_w1 AND "Unit1.Em5.ControlNodes".cm.softcam.transferPnPLeftAxisY.pos00_wait.inPos;
   #statTonTime[980].TON(IN := #_w1 AND "Unit1.Em5.ControlNodes".transferPnPLeft."step".transition1[980],
                         PT := T#100ms);
   IF #statTonTime[980].Q THEN
       "Unit1.Em5.ControlNodes".transferPnPLeft.sequence.status.nextStep := #JOB_9_STEP_81;
   END_IF;
END_REGION

REGION Network 68: Step[981] : Transfer PP Left X/Z-Axis Wait Pos
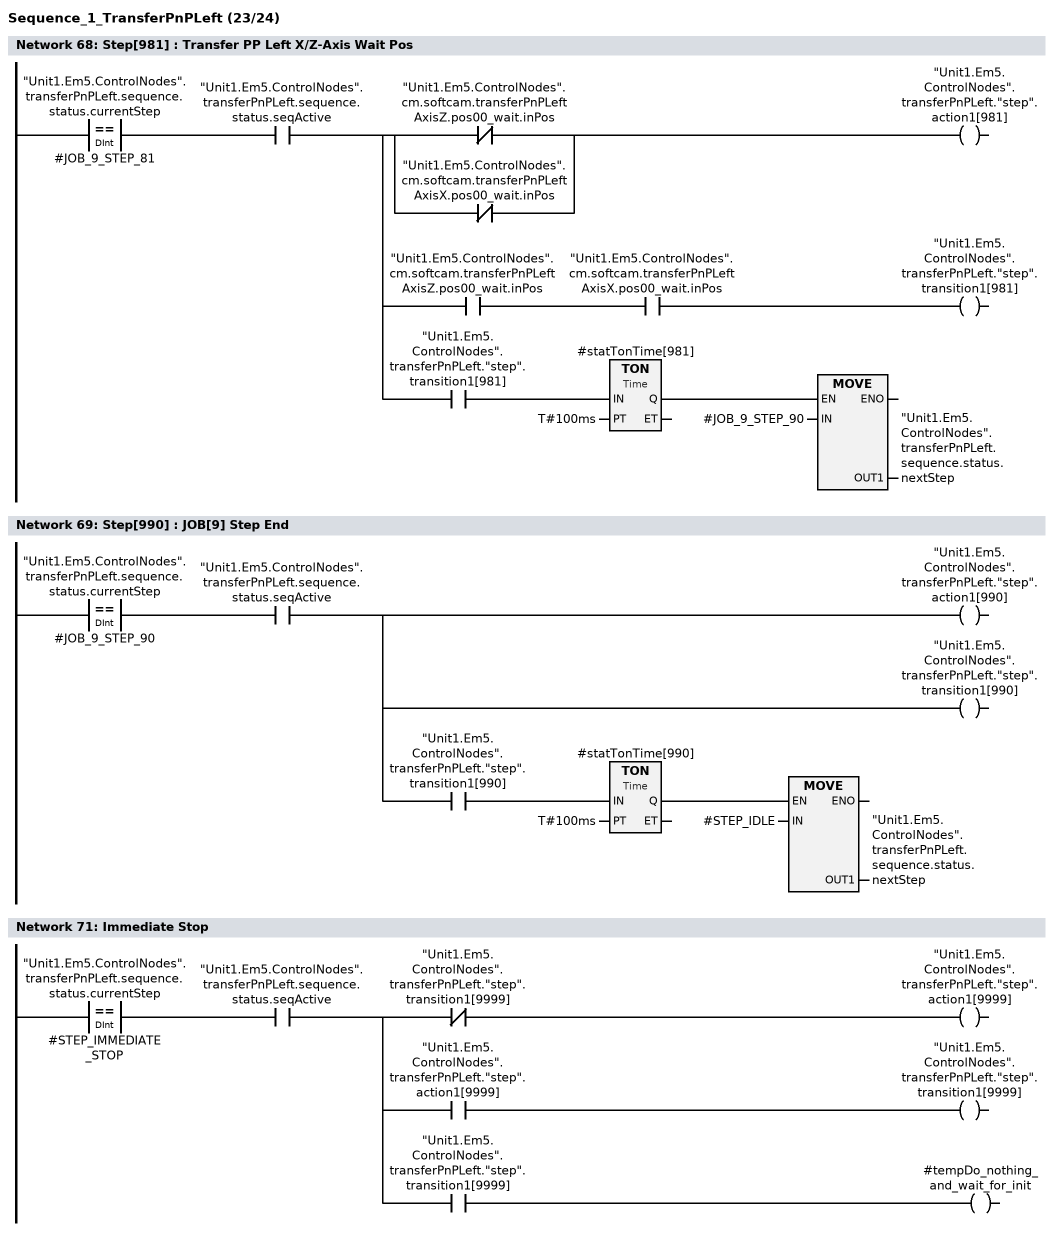
   RUNG wire#powerrail
      { S7_Templates := "SrcType := DInt" } EQ_Contact(in1 := "Unit1.Em5.ControlNodes".transferPnPLeft.sequence.status.currentStep, in2 := #JOB_9_STEP_81)
      Contact( "Unit1.Em5.ControlNodes".transferPnPLeft.sequence.status.seqActive )
      wire#w1
      I_Contact( "Unit1.Em5.ControlNodes".cm.softcam.transferPnPLeftAxisZ.pos00_wait.inPos )
      wire#w2
      Coil( "Unit1.Em5.ControlNodes".transferPnPLeft."step".action1[981] )
   END_RUNG
   RUNG wire#w1
      I_Contact( "Unit1.Em5.ControlNodes".cm.softcam.transferPnPLeftAxisX.pos00_wait.inPos )
   END_RUNG wire#w2
   RUNG wire#w1
      Contact( "Unit1.Em5.ControlNodes".cm.softcam.transferPnPLeftAxisZ.pos00_wait.inPos )
      Contact( "Unit1.Em5.ControlNodes".cm.softcam.transferPnPLeftAxisX.pos00_wait.inPos )
      Coil( "Unit1.Em5.ControlNodes".transferPnPLeft."step".transition1[981] )
   END_RUNG
   RUNG wire#w1
      Contact( "Unit1.Em5.ControlNodes".transferPnPLeft."step".transition1[981] )
      { S7_Templates := "time_type := Time" } #statTonTime[981].TON(pt := T#100ms, et =>)
      Move(in := #JOB_9_STEP_90, out1 => "Unit1.Em5.ControlNodes".transferPnPLeft.sequence.status.nextStep)
   END_RUNG
   // the same network as SCL:
   #_w1 := ("Unit1.Em5.ControlNodes".transferPnPLeft.sequence.status.currentStep = #JOB_9_STEP_81) AND "Unit1.Em5.ControlNodes".transferPnPLeft.sequence.status.seqActive;
   "Unit1.Em5.ControlNodes".transferPnPLeft."step".action1[981] := #_w1 AND (NOT "Unit1.Em5.ControlNodes".cm.softcam.transferPnPLeftAxisZ.pos00_wait.inPos OR NOT "Unit1.Em5.ControlNodes".cm.softcam.transferPnPLeftAxisX.pos00_wait.inPos);
   "Unit1.Em5.ControlNodes".transferPnPLeft."step".transition1[981] := #_w1 AND "Unit1.Em5.ControlNodes".cm.softcam.transferPnPLeftAxisZ.pos00_wait.inPos AND "Unit1.Em5.ControlNodes".cm.softcam.transferPnPLeftAxisX.pos00_wait.inPos;
   #statTonTime[981].TON(IN := #_w1 AND "Unit1.Em5.ControlNodes".transferPnPLeft."step".transition1[981],
                         PT := T#100ms);
   IF #statTonTime[981].Q THEN
       "Unit1.Em5.ControlNodes".transferPnPLeft.sequence.status.nextStep := #JOB_9_STEP_90;
   END_IF;
END_REGION

REGION Network 69: Step[990] : JOB[9] Step End
   RUNG wire#powerrail
      { S7_Templates := "SrcType := DInt" } EQ_Contact(in1 := "Unit1.Em5.ControlNodes".transferPnPLeft.sequence.status.currentStep, in2 := #JOB_9_STEP_90)
      Contact( "Unit1.Em5.ControlNodes".transferPnPLeft.sequence.status.seqActive )
      wire#w1
      Coil( "Unit1.Em5.ControlNodes".transferPnPLeft."step".action1[990] )
   END_RUNG
   RUNG wire#w1
      Coil( "Unit1.Em5.ControlNodes".transferPnPLeft."step".transition1[990] )
   END_RUNG
   RUNG wire#w1
      Contact( "Unit1.Em5.ControlNodes".transferPnPLeft."step".transition1[990] )
      { S7_Templates := "time_type := Time" } #statTonTime[990].TON(pt := T#100ms, et =>)
      Move(in := #STEP_IDLE, out1 => "Unit1.Em5.ControlNodes".transferPnPLeft.sequence.status.nextStep)
   END_RUNG
   // the same network as SCL:
   "Unit1.Em5.ControlNodes".transferPnPLeft."step".action1[990] := ("Unit1.Em5.ControlNodes".transferPnPLeft.sequence.status.currentStep = #JOB_9_STEP_90) AND "Unit1.Em5.ControlNodes".transferPnPLeft.sequence.status.seqActive;
   "Unit1.Em5.ControlNodes".transferPnPLeft."step".transition1[990] := ("Unit1.Em5.ControlNodes".transferPnPLeft.sequence.status.currentStep = #JOB_9_STEP_90) AND "Unit1.Em5.ControlNodes".transferPnPLeft.sequence.status.seqActive;
   #statTonTime[990].TON(IN := ("Unit1.Em5.ControlNodes".transferPnPLeft.sequence.status.currentStep = #JOB_9_STEP_90) AND "Unit1.Em5.ControlNodes".transferPnPLeft.sequence.status.seqActive AND "Unit1.Em5.ControlNodes".transferPnPLeft."step".transition1[990],
                         PT := T#100ms);
   IF #statTonTime[990].Q THEN
       "Unit1.Em5.ControlNodes".transferPnPLeft.sequence.status.nextStep := #STEP_IDLE;
   END_IF;
END_REGION

REGION Network 70: ******************** IMMEDIATE STOP *********************
END_REGION

REGION Network 71: Immediate Stop
   RUNG wire#powerrail
      { S7_Templates := "SrcType := DInt" } EQ_Contact(in1 := "Unit1.Em5.ControlNodes".transferPnPLeft.sequence.status.currentStep, in2 := #STEP_IMMEDIATE_STOP)
      Contact( "Unit1.Em5.ControlNodes".transferPnPLeft.sequence.status.seqActive )
      wire#w1
      I_Contact( "Unit1.Em5.ControlNodes".transferPnPLeft."step".transition1[9999] )
      Coil( "Unit1.Em5.ControlNodes".transferPnPLeft."step".action1[9999] )
   END_RUNG
   RUNG wire#w1
      Contact( "Unit1.Em5.ControlNodes".transferPnPLeft."step".action1[9999] )
      Coil( "Unit1.Em5.ControlNodes".transferPnPLeft."step".transition1[9999] )
   END_RUNG
   RUNG wire#w1
      Contact( "Unit1.Em5.ControlNodes".transferPnPLeft."step".transition1[9999] )
      Coil( #tempDo_nothing_and_wait_for_init )
   END_RUNG
   // the same network as SCL:
   #_w1 := ("Unit1.Em5.ControlNodes".transferPnPLeft.sequence.status.currentStep = #STEP_IMMEDIATE_STOP) AND "Unit1.Em5.ControlNodes".transferPnPLeft.sequence.status.seqActive;
   "Unit1.Em5.ControlNodes".transferPnPLeft."step".action1[9999] := #_w1 AND NOT "Unit1.Em5.ControlNodes".transferPnPLeft."step".transition1[9999];
   "Unit1.Em5.ControlNodes".transferPnPLeft."step".transition1[9999] := #_w1 AND "Unit1.Em5.ControlNodes".transferPnPLeft."step".action1[9999];
   #tempDo_nothing_and_wait_for_init := #_w1 AND "Unit1.Em5.ControlNodes".transferPnPLeft."step".transition1[9999];
END_REGION

REGION Network 72: ********************** STATUS **************************
END_REGION

REGION Network 73: Sequence Status
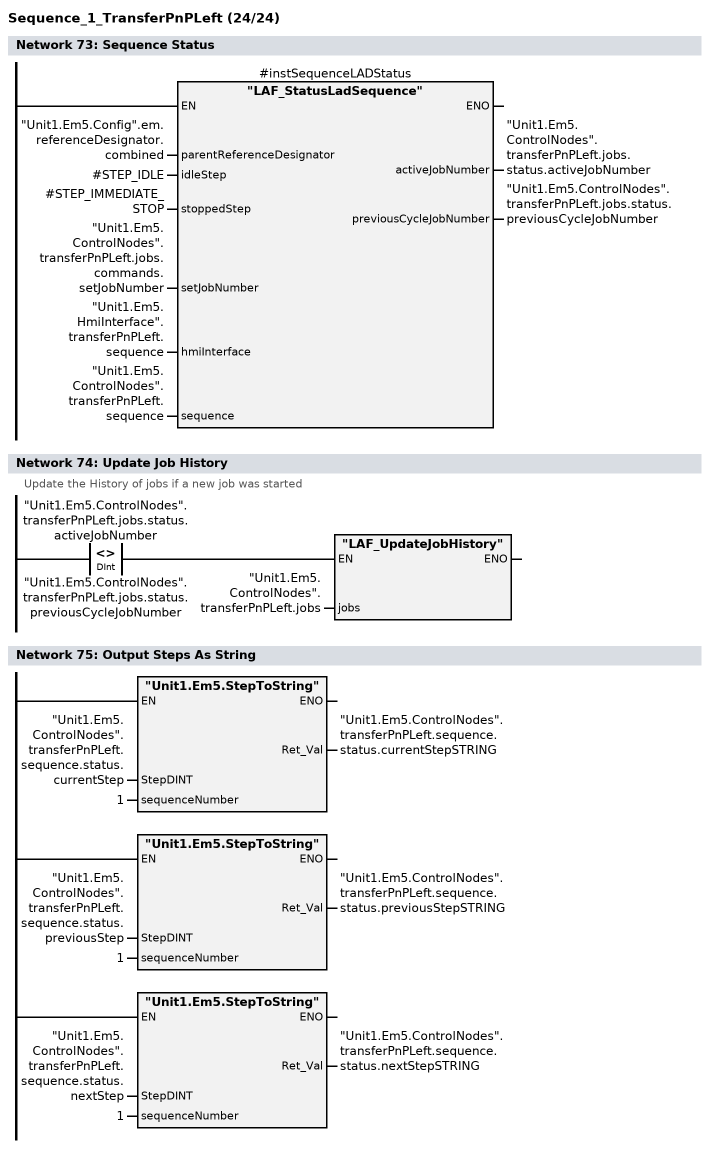
   RUNG wire#powerrail
      #instSequenceLADStatus(parentReferenceDesignator := "Unit1.Em5.Config".em.referenceDesignator.combined, idleStep := #STEP_IDLE, stoppedStep := #STEP_IMMEDIATE_STOP, setJobNumber := "Unit1.Em5.ControlNodes".transferPnPLeft.jobs.commands.setJobNumber, hmiInterface := "Unit1.Em5.HmiInterface".transferPnPLeft.sequence, sequence := "Unit1.Em5.ControlNodes".transferPnPLeft.sequence, activeJobNumber => "Unit1.Em5.ControlNodes".transferPnPLeft.jobs.status.activeJobNumber, previousCycleJobNumber => "Unit1.Em5.ControlNodes".transferPnPLeft.jobs.status.previousCycleJobNumber)
   END_RUNG
   // the same network as SCL:
   #instSequenceLADStatus(parentReferenceDesignator := "Unit1.Em5.Config".em.referenceDesignator.combined,   // "LAF_StatusLadSequence"
                          idleStep := #STEP_IDLE,
                          stoppedStep := #STEP_IMMEDIATE_STOP,
                          setJobNumber := "Unit1.Em5.ControlNodes".transferPnPLeft.jobs.commands.setJobNumber,
                          hmiInterface := "Unit1.Em5.HmiInterface".transferPnPLeft.sequence,
                          sequence := "Unit1.Em5.ControlNodes".transferPnPLeft.sequence,
                          activeJobNumber => "Unit1.Em5.ControlNodes".transferPnPLeft.jobs.status.activeJobNumber,
                          previousCycleJobNumber => "Unit1.Em5.ControlNodes".transferPnPLeft.jobs.status.previousCycleJobNumber);
END_REGION

REGION Network 74: Update Job History
   // Update the History of jobs if a new job was started
   RUNG wire#powerrail
      { S7_Templates := "SrcType := DInt" } NE_Contact(in1 := "Unit1.Em5.ControlNodes".transferPnPLeft.jobs.status.activeJobNumber, in2 := "Unit1.Em5.ControlNodes".transferPnPLeft.jobs.status.previousCycleJobNumber)
      "LAF_UpdateJobHistory"(jobs := "Unit1.Em5.ControlNodes".transferPnPLeft.jobs)
   END_RUNG
   // the same network as SCL:
   IF "Unit1.Em5.ControlNodes".transferPnPLeft.jobs.status.activeJobNumber <> "Unit1.Em5.ControlNodes".transferPnPLeft.jobs.status.previousCycleJobNumber THEN
       "LAF_UpdateJobHistory"(jobs := "Unit1.Em5.ControlNodes".transferPnPLeft.jobs);
   END_IF;
END_REGION

REGION Network 75: Output Steps As String
   RUNG wire#powerrail
      "Unit1.Em5.StepToString"(StepDINT := "Unit1.Em5.ControlNodes".transferPnPLeft.sequence.status.currentStep, sequenceNumber := 1, Ret_Val => "Unit1.Em5.ControlNodes".transferPnPLeft.sequence.status.currentStepSTRING)
   END_RUNG
   RUNG wire#powerrail
      "Unit1.Em5.StepToString"(StepDINT := "Unit1.Em5.ControlNodes".transferPnPLeft.sequence.status.previousStep, sequenceNumber := 1, Ret_Val => "Unit1.Em5.ControlNodes".transferPnPLeft.sequence.status.previousStepSTRING)
   END_RUNG
   RUNG wire#powerrail
      "Unit1.Em5.StepToString"(StepDINT := "Unit1.Em5.ControlNodes".transferPnPLeft.sequence.status.nextStep, sequenceNumber := 1, Ret_Val => "Unit1.Em5.ControlNodes".transferPnPLeft.sequence.status.nextStepSTRING)
   END_RUNG
   // the same network as SCL:
   "Unit1.Em5.ControlNodes".transferPnPLeft.sequence.status.currentStepSTRING := "Unit1.Em5.StepToString"(StepDINT := "Unit1.Em5.ControlNodes".transferPnPLeft.sequence.status.currentStep,
                           sequenceNumber := 1);
   "Unit1.Em5.ControlNodes".transferPnPLeft.sequence.status.previousStepSTRING := "Unit1.Em5.StepToString"(StepDINT := "Unit1.Em5.ControlNodes".transferPnPLeft.sequence.status.previousStep,
                           sequenceNumber := 1);
   "Unit1.Em5.ControlNodes".transferPnPLeft.sequence.status.nextStepSTRING := "Unit1.Em5.StepToString"(StepDINT := "Unit1.Em5.ControlNodes".transferPnPLeft.sequence.status.nextStep,
                           sequenceNumber := 1);
END_REGION
END_FUNCTION_BLOCK
